PROGRAM Demo
VAR

    fbMotionLogger : FB_MotionLogger;
    // Persistant storage
    fbPersistentDataStorage : FB_PersistentDataStorage;
    M1 : ST_MotionEpicsInterface;

    fbMotionStage : FB_MotionStageNC(	sName := 'NC',
                                        stMotionEpicsItf := M1,
                                        AxisRef := NcAxis_GVL.NC,
                                        iMotionLogger := fbMotionLogger,
                                        iPersistentDataStorage := fbPersistentDataStorage
                                    ) := (BrakeMode := E_StageBrakeMode.IF_MOVING, EnableMode:=ENUM_StageEnableMode.DURING_MOTION, HomeMode:=E_EpicsHomeCmd.AUTOZERO);

END_VAR

fbMotionLogger();
fbPersistentDataStorage();
fbMotionStage();

END_PROGRAM

(* stored: Version 1.1.0.1
   POU Demo: Id {61c6dfbc-a7dc-4c03-9ea3-aa217d748554}, SpecialFunc None *)
